Staubli VAL3: FACULA.pgx

public program Facula(trsf& x_trSource[], num x_nDia, num x_nType, trsf& x_trDownLead, bool& x_bRes)
  local trsf l_trTrsf
  local num l_nDia
  local num l_nNum
begin
  //光斑补偿

  if  x_nDia<=0 or x_nType==10 or x_nType==9
     x_bRes=true
     return
  endIf

  //光斑强制设置为0.1
  if x_nDia>1
    x_nDia=0.1
  endIf


  if x_nType==2
    x_trDownLead.ry=max(x_trDownLead.ry-x_nDia,0.1)
    x_bRes=true
    return
  endIf

  if x_nType==12
    x_trDownLead.ry=x_trDownLead.ry+x_nDia
    x_bRes=true
    return
  endIf

  l_nDia=0

  call Circumcircle(x_trSource,l_trTrsf,l_nDia,x_bRes)
  if !x_bRes
    return
  endIf

  if x_nDia>=l_nDia/2
    x_nDia=0
    x_bRes=true
    return
  endIf


  switch x_nType
    case 1,3,4,5,6,7,8

      l_nDia=l_nDia-x_nDia*2
    break

    case 11,13,14,15,16,17,18
      l_nDia=l_nDia+x_nDia*2

    break

  endSwitch


  call ChangeCpoint(x_trSource,l_nDia,x_bRes)

end
